TYPE E_Payload_Type :
(
	NO_PAYLOAD := 0,
	PAYLOAD_A,
	PAYLOAD_B,
	SYNCH_PAYLOAD,
	PAYLOAD_TYPE_SIZE
);
END_TYPE

(* stored: Version 1.1.0.1, ProductVersion 3.1.4024.2
   DUT E_Payload_Type: Id {0a0887d1-1dfe-4f14-b27b-0145f54e5547} *)
